// TwinCAT 3 PLC project Magnet_Measurement
// ProgramVersion: 3.1.4023.0
// libraries:
//   CmpBitmapPool, * (System)
//   Tc2_ControllerToolbox, * (Beckhoff Automation GmbH)
//   Tc2_Database, * (Beckhoff Automation GmbH)
//   Tc2_Standard, * (Beckhoff Automation GmbH)
//   Tc2_System, * (Beckhoff Automation GmbH)
//   Tc2_Utilities, * (Beckhoff Automation GmbH)
//   Tc3_Database, * (Beckhoff Automation GmbH)
//   Tc3_EventLogger, * (Beckhoff Automation GmbH)
//   Tc3_Module, * (Beckhoff Automation GmbH)
//   VisuDialogs, * (System)
//   VisuSymbols,3.5.10.0,System
// project tree:
//   DUTs/ ST_Data.TcDUT, ST_HMI_Plot_Array.TcDUT, ST_Masurdata.TcDUT, ST_Metadata.TcDUT
//   / GlobalTextList.TcGTLO, PlcTask.TcTTO, Visualisierungsmanager.TcVMO (not stored)
//   GVLs/ GVL_masur.TcGVL, GVL_IO.TcGVL, GVL_Meta.TcGVL
//   POUs/ FB_Write_Metadata.TcPOU, Log_Data_Buffer.TcPOU
//   VISUs/ GVL_Visu.TcGVL, ImagePool.TcIPO (not stored), Startpage.TcVIS, Write_Metadata_Visu.TcVIS, Visualization.TcVIS
// real-time tasks:
//   TASK PlcTask: cycle T#20ms, priority 20, ADS port 350
// I/O:
//   DEVICE Gerät 1 (EtherCAT) (disabled), AmsNetId 192.168.56.1.2.1
//     Box 1 (BK1120)

CONFIGURATION Magnet_Measurement
    RESOURCE PLC ON TwinCAT3
        TASK PlcTask(INTERVAL := T#20ms, PRIORITY := 20);
        PROGRAM Log_Data_Buffer WITH PlcTask : Log_Data_Buffer;
    END_RESOURCE
END_CONFIGURATION

// ---- DUTs/ST_Data.TcDUT
TYPE ST_Data :
STRUCT
	power: REAL;
	test: REAL;
	timestamp: REAL;
END_STRUCT
END_TYPE

// ---- DUTs/ST_HMI_Plot_Array.TcDUT
TYPE ST_HMI_Plot_Array :
STRUCT
	x : REAL := 0;
	y : REAL := 0;
END_STRUCT
END_TYPE

// ---- DUTs/ST_Masurdata.TcDUT
TYPE ST_Masurdata :
STRUCT
	id: INT;
	time2: REAL;
	primary_power: REAL;
	secondary_power: REAL;
	phase_shift: REAL;
	frequency: REAL;
	flux_density: REAL;
	Meta_id: INT;
END_STRUCT
END_TYPE

// ---- DUTs/ST_Metadata.TcDUT
TYPE ST_Metadata :
STRUCT
	Id: LINT;
	measurementname: STRING(255);
	carried_out: STRING(255);
	thickness: REAL;
	steel: STRING(255);
	joint_pre: STRING(255);
	root_face: REAL;
	opening_angel: REAL;
	edge_pre: STRING(255);
	welding_speed: REAL;
	laser_power: REAL;
	focal_position: REAL;
	distance_a_l: REAL;
	wire_feeding_rate: REAL;
	wire_diameter: REAL;
	wire_type: STRING(255);
	stickout: REAL;
	arc_dynamic: REAL;
	frequency: REAL;
	voltage_ac_power_source: REAL;
	distance_magnet_pole: REAL;
	magnet_pole_width: REAL;
	magnet_pole_type: STRING(255);
	core_dimension: REAL;
	very_good: STRING(255);
	normal: STRING(255);
	uniform_root_overcome: STRING(255);
	undercut: STRING(255);
	sporadic_seam_collapse: STRING(255);
	sporadic_dropout: STRING(255);
	bad: STRING(255);
	periodic_dropout: STRING(255);
	strong_seam_collapse: STRING(255);
	incomplite_penetration: STRING(255);
END_STRUCT
END_TYPE

// ---- GVLs/GVL_masur.TcGVL
{attribute 'qualified_only'}
VAR_GLOBAL
	id : INT; //wird automatisch erstellt
	time2 : REAL;
	primary_power: REAL;
	secondary_power: REAL;
	phase_shift: REAL;
	frequency: REAL;
	flux_density: REAL;
	Meta_id: INT;
END_VAR

// ---- GVLs/GVL_IO.TcGVL
{attribute 'qualified_only'}
VAR_GLOBAL
	//Raw data read every cycle
	//Primärspule
	gl_voltage_effective_raw_prime AT %I* : UINT := 15000; //Effektivwert Spannung Primärspule Rohwert
	gl_voltage_periode_raw_prime AT  %I* : UINT := 20; //Periode Spannungsignal Primärspule Rohwert
	gl_current_effective_raw_prime AT %I* : UINT := 3800; //Effektivwert Stromstärke Primärspule Rohwert
	gl_current_periode_raw_prime AT %I* : UINT := 20; //Periode Stromstärkesignal Primärspule Rohwert
	//Sekundärspule
	gl_voltage_effective_raw_secondary AT %I* : UINT := 20546; //Effektivwert Spannung Sekundärspule Rohwert
	gl_voltage_periode_raw_secondary AT  %I* : UINT := 20; //Periode Spannungsignal Sekundärspule Rohwert
	gl_current_effective_raw_secondary AT %I* : UINT := 3800; //Effektivwert Stromstärke Sekundärspule Rohwert
	gl_current_periode_raw_secondary AT %I* : UINT := 20; //Periode Stromstärkesignal Sekundärspule Rohwert
END_VAR

// ---- GVLs/GVL_Meta.TcGVL
{attribute 'qualified_only'}
VAR_GLOBAL
	// Variablen for Database Metadata Table
	Id : LINT := 11; //wird automatisch erstellt beim schreiben
	measurementname: STRING(255) := 'test';
	carried_out: STRING(255) := 'test1';
	thickness: REAL := 1;
	steel: STRING(255) := 'stahl';
	joint_pre: STRING(255) := 'squer';
	root_face: REAL := 0;
	opening_angel: REAL := 0;
	edge_pre: STRING(255) := 'aet';
	welding_speed: REAL := 0;
	laser_power: REAL := 1;
	focal_position: REAL := 2;
	distance_a_l: REAL := 3;
	wire_feeding_rate: REAL := 4;
	wire_diameter: REAL := 5;
	wire_type: STRING(255) := 'tea';
	stickout: REAL := 6;
	arc_dynamic: REAL := 2;
	frequency: REAL := 1;
	voltage_ac_power_source: REAL := 22;
	distance_magnet_pole: REAL := 33;
	magnet_pole_width: REAL := 22;
	magnet_pole_type: STRING(255) := 'at';
	core_dimension: REAL := 22;
	very_good: STRING(255) := 'asd';
	normal: STRING(255) := 'asd';
	uniform_root_overcome: STRING(255) := 'asd';
	undercut: STRING(255) := 'asdw';
	sporadic_seam_collapse: STRING(255) := 'aaa';
	sporadic_dropout: STRING(255) := 'aw';
	bad: STRING(255) := 'aaaw';
	periodic_dropout: STRING(255) := 'asdaw';
	strong_seam_collapse: STRING(255) := 'aqqq';
	incomplite_penetration: STRING(255) := 'öpkl';
END_VAR

// ---- VISUs/GVL_Visu.TcGVL
{attribute 'qualified_only'}
VAR_GLOBAL
	start_record : BOOL := FALSE;
END_VAR

// ---- POUs/Log_Data_Buffer.TcPOU
PROGRAM Log_Data_Buffer
VAR
	//Messvariablen
	voltage_effective_prime : REAL; //Effektivwert Spannung Primärspule umgewandelt auf +-10V
	voltage_frequency_prime : REAL; //Frequenz Primärspule Spannungssignal umgewandelt auf +-10 in Hz
	current_effective_prime : REAL; //Effektivwert Stromstärke Primärspule umgewandelt auf +-10V umgewandelt zu Ampere
	current_frequency_prime : REAL; //Frequenz Primärspule Stromstärkesignal umgewandelt auf +-10 Hz
	voltage_effective_secondary : REAL; //Effektivwert Spannung Sekundärspule umgewandelt auf +-10V
	voltage_frequency_secondary : REAL; //Frequenz Sekundärspule Spannungssignal umgewandelt auf +-10 Hz
	current_effective_secondary : REAL; //Effektivwert Stromstärke Sekundärspule umgewandelt auf +-10V umgewandelt zu Ampere
	current_frequency_secondary : REAL; //Frequenz Sekundärspule Stromstärkesignal umgewandelt auf +-10 Hz
	power_prime : REAL; //Leistung Primärspule W
	power_secondary : REAL; //Leistung Sekundärspule W
    
	//Arrays zum Plotten für HMI
	power_hmi_array : ARRAY[1..2,1..100] OF ST_HMI_Plot_Array;
	//power_secondary_hmi_array : ARRAY[1..1,1..100] OF ST_HMI_Plot_Array;
	i : INT := 1;
    rand : DRAND; 
    nrand: LREAL;
	
	fbGetCurTaskIdx  : GETCURTASKINDEX;
    ncycletime       : REAL;
	nState: INT;	
	bRecord : BOOL;
	//for generating timestamp
	fbGetSystemTime1: GetSystemTime;
	dwTimeLoDW: DWORD;
	dwTimeHiDW: DWORD;
	tFileTime: T_FILETIME;
	nTimestamp: REAL;
	//for insert meta data
	fbWriteMetadata : FB_Write_Metadata;
	fb_Start_Log : FB_PLCDBAutoLogEvt (sNetID:='', tTimeout := T#1S);
	write_meta : BOOL;
	write_meta_status : BOOL; 
	write_meta_error : BOOL; 
	meta_data_written_index : INT := 1;
	
	//for insert masur samples
	fbPLCDBCmd: FB_PLCDBCmdEvt(sNetID:= '', tTimeout:= T#19S);
	aPara: ARRAY [0..7] OF ST_ExpParameter;	
	sCmd1: STRING(255);
	sCmd2: STRING(255);
	sCmd: STRING(512); //CONCAT of sCmd1 and sCmd2
	
	//Data buffer for masur data
	aWriteSQL: ARRAY [0..19] OF BOOL;
	stData: ARRAY [0..19,0..99] OF ST_Masurdata;
	
	//buffer index and masur data variables
	nWriteBufferIndex: INT := 0;
	nWriteIndex: INT := 0;
	nSQLIndex: INT := 0;					
	bError: BOOL;
	bTableCreated: BOOL;
	bRecording: BOOL;
	nRecords: INT;
	sTableName: T_MaxString := 'masur';
	nDBID: UDINT := 1;
	timestampp : REAL := 0;
	index : INT := 0;
	id: INT := 1852;
	
	// Eventlogger
	ipTcResult: Tc3_Database.I_TcMessage;

END_VAR

// Convert Data and get the raw data
//Primärspule
rand();
nrand := rand.Num;
voltage_effective_prime := UINT_TO_REAL(GVL_IO.gl_voltage_effective_raw_prime)/65535*20; //Map UINT range of 0:65535 to +-10V 
voltage_frequency_prime := 1/(UINT_TO_REAL(GVL_IO.gl_voltage_periode_raw_prime)/1000); //convert ms to S and get Frequency from Period
current_effective_prime := UINT_TO_REAL(GVL_IO.gl_current_effective_raw_prime)/65535*20; //Map UINT range of 0:65535 to +-10V 
current_frequency_prime := 1/(UINT_TO_REAL(GVL_IO.gl_current_periode_raw_prime)/1000); //convert ms to S and get Frequency from Period
power_prime := voltage_effective_prime * current_effective_prime + nrand/3;
//Sekundärspule
voltage_effective_secondary := UINT_TO_REAL(GVL_IO.gl_voltage_effective_raw_secondary)/65535*20; //Map UINT range of 0:65535 to +-10V 
voltage_frequency_secondary := 1/(UINT_TO_REAL(GVL_IO.gl_voltage_periode_raw_secondary)/1000); //convert ms to S and get Frequency from Period
current_effective_secondary := UINT_TO_REAL(GVL_IO.gl_current_effective_raw_secondary)/65535*20; //Map UINT range of 0:65535 to +-10V 
current_frequency_secondary := 1/(UINT_TO_REAL(GVL_IO.gl_current_periode_raw_secondary)/1000); //convert ms to S and get Frequency from Period
power_secondary := voltage_effective_secondary * current_effective_secondary + nrand/2;

fbGetCurTaskIdx();
ncycletime := _TaskInfo[fbGetCurTaskIdx.index].CycleTime/10000;

//HMI Plot Array befüllen
IF (i <= 100) THEN
	//power_prime_hmi_array[1,i].x := i*ncycletime;
	//power_prime_hmi_array[1,i].y := power_prime;
	//power_secondary_hmi_array[1,i].x := i*ncycletime;
	//power_secondary_hmi_array[1,i].y := power_secondary;
	power_hmi_array[1,i].x := i*ncycletime;
	power_hmi_array[1,i].y := power_prime;
	power_hmi_array[2,i].x := i*ncycletime;
	power_hmi_array[2,i].y := power_secondary;
	i := i +1;
	ELSE
		i := 1;
END_IF
//FOR i := 1 TO 100 DO
//	power_prime_hmi_array[1,i].x := i;
//	power_prime_hmi_array[1,i].x := i;
//END_FOR//

//Create timestamp
fbGetSystemTime1(timeLoDW=>dwTimeLoDW,timeHiDW=>dwTimeHiDW);
tFileTime.dwLowDateTime := dwTimeLoDW;
tFileTime.dwHighDateTime := dwTimeHiDW;	
MEMCPY(ADR(nTimestamp), ADR(tFileTime), 8);

CASE nState OF
	0://Init
		IF bRecord THEN			
			bError := FALSE;
			bRecording := FALSE;
			nRecords := 0;
			//sTableName := 'Magnet';//CONCAT('tbl_TestSignals_', LINT_TO_STRING(nTimestamp)); //create new tablename
			sCmd1 := CONCAT('INSERT INTO ', sTableName);
			sCmd2 := ' ([id],[time2],[primary_power],[secondary_power],[phase_shift],[frequency],[flux_density],[Meta_id]) VALUES({id},{time2},{primary_power},{secondary_power},{phase_shift},{frequency},{flux_density},{Meta_id});';
			CONCAT2(ADR(sCmd1), ADR(sCmd2), ADR(sCmd), SIZEOF(sCmd));
			
			aPara[0].sParaName:= 'id'; 				aPara[0].nParaSize:= 8; 	aPara[0].eParaType:= E_ExpParameterType.Int32 ;
			aPara[1].sParaName:= 'time2'; 			aPara[1].nParaSize:= 8; 	aPara[1].eParaType:= E_ExpParameterType.Float32 ;		
			aPara[2].sParaName:= 'primary_power';	aPara[2].nParaSize:= 8;		aPara[2].eParaType:= E_ExpParameterType.Float32 ;		
			aPara[3].sParaName:= 'secondary_power';	aPara[3].nParaSize:= 8;		aPara[3].eParaType:= E_ExpParameterType.Float32 ;	
			aPara[4].sParaName:= 'phase_shift';		aPara[4].nParaSize:= 8;		aPara[4].eParaType:= E_ExpParameterType.Float32 ;
			aPara[5].sParaName:= 'frequency';		aPara[5].nParaSize:= 8;		aPara[5].eParaType:= E_ExpParameterType.Float32 ;
			aPara[6].sParaName:= 'flux_density';	aPara[6].nParaSize:= 8;		aPara[6].eParaType:= E_ExpParameterType.Float32 ;
			aPara[7].sParaName:= 'Meta_id';			aPara[7].nParaSize:= 8;		aPara[7].eParaType:= E_ExpParameterType.Int32 ;	
			nWriteBufferIndex := 0;
			nWriteIndex := 0;
			nSQLIndex := 0;	
			nState := 1;
		END_IF
		
	1://Idle
		IF write_meta THEN
			IF meta_data_written_index = 1 THEN
				fb_Start_Log.RunOnce(hAutologGrpID := 1, bAll := TRUE);
				meta_data_written_index := 2;
			ELSE 
				fb_Start_Log.RunOnce(hAutologGrpID := 1, bAll := TRUE);
				fb_Start_Log.RunOnce(hAutologGrpID := 1, bAll := TRUE);
				fb_Start_Log.RunOnce(hAutologGrpID := 1, bAll := TRUE);
			END_IF
			write_meta := FALSE;
			write_meta_status := fb_Start_Log.bBusy;
			write_meta_error := fb_Start_Log.bError;
		END_IF
		
	2://Recording		
		bRecording := TRUE;
		//Fill buffer
		stData[nWriteBufferIndex, nWriteIndex].id := id;
		stData[nWriteBufferIndex, nWriteIndex].time2 := timestampp;
		stData[nWriteBufferIndex, nWriteIndex].primary_power := power_prime;
		stData[nWriteBufferIndex, nWriteIndex].secondary_power := power_secondary;
		stData[nWriteBufferIndex, nWriteIndex].phase_shift := 1.0;
		stData[nWriteBufferIndex, nWriteIndex].frequency := 2.0;
		stData[nWriteBufferIndex, nWriteIndex].flux_density := 3.0;
		stData[nWriteBufferIndex, nWriteIndex].Meta_id := 1;
		timestampp := ncycletime * index;
		index := index + 1;
		id := id + 1;
		//Set buffer index
		nWriteIndex := nWriteIndex + 1;		
		IF nWriteIndex = 100 THEN
			nWriteIndex := 0;
			aWriteSQL[nWriteBufferIndex]:= TRUE;
			nWriteBufferIndex := nWriteBufferIndex + 1;
			
			IF nWriteBufferIndex = 20 THEN
				nWriteBufferIndex := 0;
			END_IF 	
			
			IF aWriteSQL[nWriteBufferIndex] THEN
				nState := 255;
				RETURN;
			END_IF
		END_IF
				
		//Write buffer element (100 samples) to database
		IF aWriteSQL[nSQLIndex] THEN
			ipTcResult := fbPLCDBCmd.ipTcResult;
			IF fbPLCDBCmd.Execute(nDBID, ADR(sCmd), SIZEOF(sCmd), ADR(stData[nSQLIndex,0]), SIZEOF(stData[nSQLIndex,0]) * 100, ADR(aPara), SIZEOF(aPara)) THEN
				IF fbPLCDBCmd.bError THEN					
					nState := 255;
				ELSE
					nRecords := nRecords + 100;
					
					aWriteSQL[nSQLIndex] := FALSE;
					
					nSQLIndex := nSQLIndex + 1;
					IF nSQLIndex = 20 THEN
						nSQLIndex := 0;
					END_IF
					
					IF NOT bRecord THEN
						bRecording := FALSE;
						nState := 0;
					END_IF
				END_IF				
			END_IF
		END_IF
		
	255://Error
		bError := TRUE;
		bRecording := FALSE;
		IF NOT bRecord THEN			
			nState := 0;
		END_IF 
END_CASE

END_PROGRAM

// ---- POUs/FB_Write_Metadata.TcPOU
FUNCTION_BLOCK FB_Write_Metadata
VAR
	stMetadata : ST_Metadata;
	//fbPLCWrite : FB_PLCDBWriteEvt(sNetID:='', tTimeout:=T#15S);
	//arrColumns: ARRAY[0..33] OF STRING(255) := ['Id', 'measurementname', 'carried_out', 'thickness', 'steel', 'joint_pre', 'root_face', 'opening_angel', 'edge_pre', 'welding_speed', 'laser_power', 'focal_position', 'distance_a_l', 'wire_feeding_rate', 'wire_diameter', 'wire_type', 'stickout', 'arc_dynamic', 'frequency', 'voltage_ac_power_source', 'distance_magnet_pole', 'magnet_pole_width', 'magnet_pole_type', 'core_dimension', 'very_good', 'normal', 'uniform_root_overcome', 'undercut', 'sporadic_seam_collapse', 'sporadic_dropout', 'bad', 'periodic_dropout', 'strong_seam_collapse', 'incomplite_penetration'];
	stData123 : ST_Data;
	fb_PLCDBWriteEvt: FB_PLCDBWriteEvt(sNetID:='', tTimeout:=T#5S);
	arrColumns: ARRAY [0..2] OF STRING(50) := ['power', 'test', 'timestamp'];
	
END_VAR
VAR_OUTPUT
	status : BOOL;
END_VAR

// Get variables from global list form Visu Interface 
stMetadata.Id := GVL_Meta.Id;
stMetadata.measurementname := GVL_Meta.measurementname;
stMetadata.carried_out := GVL_Meta.carried_out;
stMetadata.thickness := GVL_Meta.thickness;
stMetadata.steel := GVL_Meta.steel;
stMetadata.joint_pre := GVL_Meta.joint_pre;
stMetadata.root_face := GVL_Meta.root_face;
stMetadata.opening_angel := GVL_Meta.opening_angel;
stMetadata.edge_pre := GVL_Meta.edge_pre;
stMetadata.welding_speed := GVL_Meta.welding_speed;
stMetadata.laser_power := GVL_Meta.laser_power;
stMetadata.focal_position := GVL_Meta.focal_position;
stMetadata.distance_a_l := GVL_Meta.distance_a_l;
stMetadata.wire_feeding_rate := GVL_Meta.wire_feeding_rate;
stMetadata.wire_diameter := GVL_Meta.wire_diameter;
stMetadata.wire_type := GVL_Meta.wire_type;
stMetadata.stickout := GVL_Meta.stickout;
stMetadata.arc_dynamic := GVL_Meta.arc_dynamic;
stMetadata.frequency := GVL_Meta.frequency;
stMetadata.voltage_ac_power_source := GVL_Meta.voltage_ac_power_source;
stMetadata.distance_magnet_pole := GVL_Meta.distance_magnet_pole;
stMetadata.magnet_pole_width := GVL_Meta.magnet_pole_width;
stMetadata.magnet_pole_type := GVL_Meta.magnet_pole_type;
stMetadata.core_dimension := GVL_Meta.core_dimension;
stMetadata.very_good := GVL_Meta.very_good;
stMetadata.normal := GVL_Meta.normal;
stMetadata.uniform_root_overcome := GVL_Meta.uniform_root_overcome;
stMetadata.undercut := GVL_Meta.undercut;
stMetadata.sporadic_seam_collapse := GVL_Meta.sporadic_seam_collapse;
stMetadata.sporadic_dropout := GVL_Meta.sporadic_dropout;
stMetadata.bad := GVL_Meta.bad;
stMetadata.periodic_dropout := GVL_Meta.periodic_dropout;
stMetadata.strong_seam_collapse := GVL_Meta.strong_seam_collapse;
stMetadata.incomplite_penetration := GVL_Meta.incomplite_penetration;

//Test
stData123.power := 1.0;
stData123.test := 2.0;
stData123.timestamp := 3.0;
//IF NOT fb_PLCDBWriteEvt.bBusy THEN
	fb_PLCDBWriteEvt.WriteStruct(
			hDBID:= 1, 
			sTableName:= 'Magnet', 
			pRecord:= ADR(stData123), 
			cbRecord:= SIZEOF(stData123), 
			pColumnNames:= ADR(arrColumns), 
			cbColumnNames:= SIZEOF(arrColumns));
//END_IF

//write struct with event to database table Meta
//IF NOT fbPLCWrite.bBusy THEN
//	fbPLCWrite.WriteStruct(
//	hDBID:= 1, 
//	sTableName:= 'Meta', 
//	pRecord:= ADR(stMetadata), 
//	cbRecord:= SIZEOF(stMetadata), 
//	pColumnNames:= ADR(arrColumns), 
//	cbColumnNames:= SIZEOF(arrColumns));
//END_IF

//IF fbPLCWrite.bError THEN
//	status := TRUE;
//ELSE
//	status := FALSE;	
//END_IF

END_FUNCTION_BLOCK

// ---- GlobalTextList.TcGTLO
TEXTLIST GlobalTextList
  699 = '%f'
  92 = '%i'
  962 = '%s'
  908 = 'Arc Dynamic'
  755 = 'Bad'
  149 = 'Carried Out'
  470 = 'Core Dimension'
  79 = 'Distance a_l'
  864 = 'Distance Magnet Pole'
  103 = 'dtj'
  832 = 'Edge Pre'
  480 = 'est'
  342 = 'Focal Position'
  478 = 'Frequency'
  55 = 'ID'
  734 = 'Incomplete Penetration'
  457 = 'Joint Pre'
  502 = 'Laser Power'
  766 = 'Magent Pole Type'
  266 = 'Magnet Measurement HMI'
  930 = 'Magnet Pole Width'
  422 = 'Measurement\t Name'
  335 = 'Measurement Name'
  56 = 'Measurementname'
  340 = 'Measurmentname'
  418 = 'Normal'
  193 = 'Opening Angel'
  887 = 'Periodic Dopout'
  9 = 'Root Face'
  388 = 'Root Opening Angel'
  257 = 'Sporadic Dropout'
  200 = 'Sporadic Seam Collapse'
  327 = 'Start PLC Connection'
  42 = 'Status'
  144 = 'Statusword'
  188 = 'Steel'
  46 = 'Stickout'
  650 = 'Strong Seam Collapse'
  230 = 'Thickness'
  58 = 'Undercut'
  974 = 'Uniform Root Overcome'
  95 = 'Very Good'
  336 = 'Voltafage AC Power Source'
  711 = 'Voltage AC Power Source'
  745 = 'Voltatage AC Power Source'
  341 = 'Welding Speed'
  262 = 'WER'
  106 = 'Wire Diameter'
  270 = 'Wire Feeding Rate'
  572 = 'Wire Type'
  182 = 'Write Metadata'
END_TEXTLIST

// ---- VISUs/Startpage.TcVIS
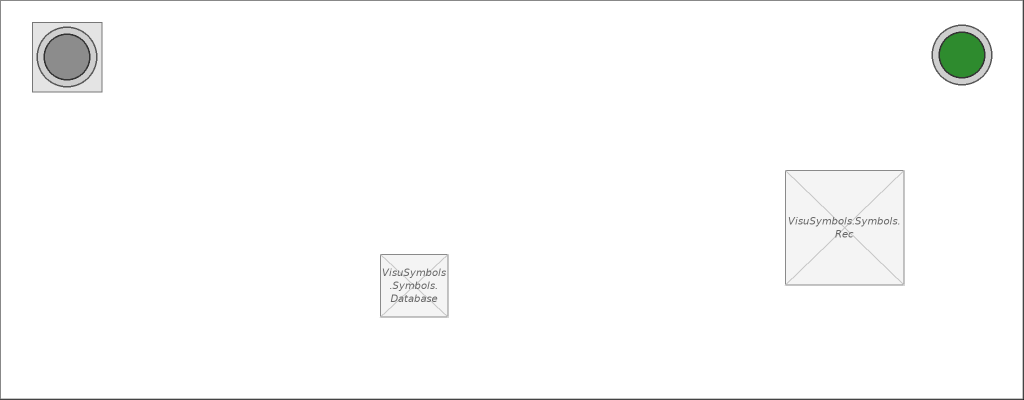
VISUALIZATION Startpage  // 1024x400
    RoundedRectangle (0,0 1024x400)
    PushSwitchLed (32,22 70x70), behaviour: TOGGLE, style: Switch-PushSwitchLed-Gray
    Lamp1 (927,20 70x70), style: Lamp-Lamp1-Green
    Image (785,170 119x115), image: VisuSymbols.Symbols.Rec
    Image (380,254 68x63), image: VisuSymbols.Symbols.Database
END_VISUALIZATION

// ---- VISUs/Write_Metadata_Visu.TcVIS
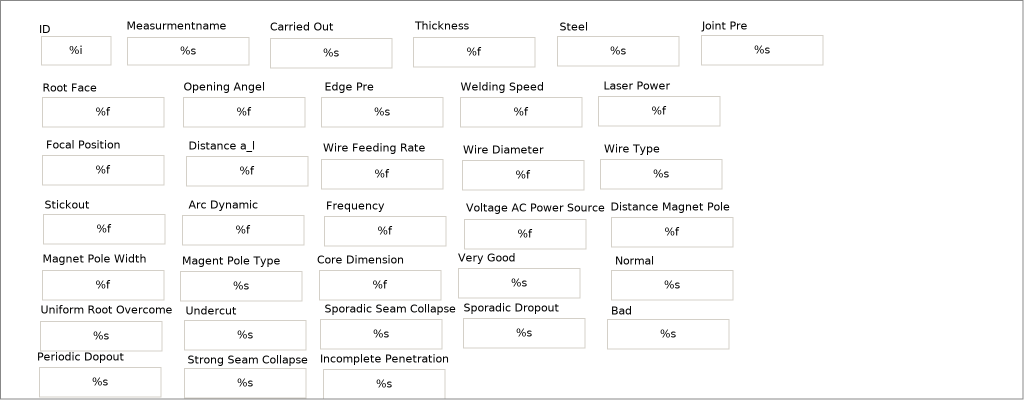
VISUALIZATION Write_Metadata_Visu  // 1024x400
    Textfield (41,36 70x29), "%i", text variable: GVL_Meta.Id
        OnMouseDown: write the text variable via Default
    Label (10,15 70x29), "ID"
    Textfield (127,37 122x28), "%s", text variable: GVL_Meta.measurementname
        OnMouseClick: write the text variable via Default
    Label (117,13 119x26), "Measurmentname"
    Textfield (270,38 122x30), "%s", text variable: GVL_Meta.Id
        OnMouseClick: write the text variable via Default
    Label (264,13 76x28), "Carried Out"
    Textfield (413,37 122x30), "%f", text variable: GVL_Meta.thickness
        OnMouseClick: write the text variable via Default
    Label (404,12 76x28), "Thickness"
    Textfield (557,36 122x30), "%s", text variable: GVL_Meta.steel
        OnMouseClick: write the text variable via Default
    Label (545,13 58x28), "Steel"
    Textfield (701,35 122x30), "%s", text variable: GVL_Meta.joint_pre
        OnMouseClick: write the text variable via Default
    Label (696,12 58x28), "Joint Pre"
    Textfield (42,97 122x30), "%f", text variable: GVL_Meta.root_face
        OnMouseClick: write the text variable via Default
    Label (41,74 58x28), "Root Face"
    Textfield (183,97 122x30), "%f", text variable: GVL_Meta.opening_angel
        OnMouseClick: write the text variable via Default
    Label (167,73 115x28), "Opening Angel"
    Textfield (321,97 122x30), "%s", text variable: GVL_Meta.edge_pre
        OnMouseClick: write the text variable via Default
    Label (316,73 67x28), "Edge Pre"
    Textfield (460,97 122x30), "%f", text variable: GVL_Meta.welding_speed
        OnMouseClick: write the text variable via Default
    Label (451,73 103x28), "Welding Speed"
    Textfield (598,96 122x30), "%f", text variable: GVL_Meta.laser_power
        OnMouseClick: write the text variable via Default
    Label (588,72 98x28), "Laser Power"
    Textfield (42,155 122x30), "%f", text variable: GVL_Meta.focal_position
        OnMouseClick: write the text variable via Default
    Label (26,131 115x28), "Focal Position"
    Textfield (186,156 122x30), "%f", text variable: GVL_Meta.distance_a_l
        OnMouseClick: write the text variable via Default
    Label (173,132 98x28), "Distance a_l"
    Textfield (321,159 122x30), "%f", text variable: GVL_Meta.wire_feeding_rate
        OnMouseClick: write the text variable via Default
    Label (317,134 115x28), "Wire Feeding Rate"
    Textfield (462,160 122x30), "%f", text variable: GVL_Meta.wire_diameter
        OnMouseClick: write the text variable via Default
    Label (446,136 115x28), "Wire Diameter"
    Textfield (600,159 122x30), "%s", text variable: GVL_Meta.wire_type
        OnMouseClick: write the text variable via Default
    Label (589,135 86x28), "Wire Type"
    Textfield (43,214 122x30), "%f", text variable: GVL_Meta.stickout
        OnMouseClick: write the text variable via Default
    Label (33,191 68x28), "Stickout"
    Textfield (182,215 122x30), "%f", text variable: GVL_Meta.arc_dynamic
        OnMouseClick: write the text variable via Default
    Label (166,191 115x28), "Arc Dynamic"
    Textfield (324,216 122x30), "%f", text variable: GVL_Meta.frequency
        OnMouseClick: write the text variable via Default
    Label (298,192 115x28), "Frequency"
    Textfield (464,219 122x30), "%f", text variable: GVL_Meta.voltage_ac_power_source
        OnMouseClick: write the text variable via Default
    Label (454,194 163x28), "Voltage AC Power Source"
    Textfield (611,217 122x30), "%f", text variable: GVL_Meta.distance_magnet_pole
        OnMouseClick: write the text variable via Default
    Label (603,193 135x28), "Distance Magnet Pole"
    Textfield (42,270 122x30), "%f", text variable: GVL_Meta.magnet_pole_width
        OnMouseClick: write the text variable via Default
    Label (37,245 115x28), "Magnet Pole Width"
    Textfield (180,271 122x30), "%s", text variable: GVL_Meta.magnet_pole_type
        OnMouseClick: write the text variable via Default
    Label (174,247 115x28), "Magent Pole Type"
    Textfield (319,270 122x30), "%f", text variable: GVL_Meta.core_dimension
        OnMouseClick: write the text variable via Default
    Label (303,246 115x28), "Core Dimension"
    Textfield (458,268 122x30), "%s", text variable: GVL_Meta.very_good
        OnMouseClick: write the text variable via Default
    Label (440,244 94x28), "Very Good"
    Textfield (611,270 122x30), "%s", text variable: GVL_Meta.normal
        OnMouseClick: write the text variable via Default
    Label (601,247 67x28), "Normal"
    Textfield (40,321 122x30), "%s", text variable: GVL_Meta.uniform_root_overcome
        OnMouseClick: write the text variable via Default
    Label (32,296 149x28), "Uniform Root Overcome"
    Textfield (184,320 122x30), "%s", text variable: GVL_Meta.undercut
        OnMouseClick: write the text variable via Default
    Label (172,297 78x28), "Undercut"
    Textfield (320,319 122x30), "%s", text variable: GVL_Meta.sporadic_seam_collapse
        OnMouseClick: write the text variable via Default
    Label (315,295 151x28), "Sporadic Seam Collapse"
    Textfield (463,318 122x30), "%s", text variable: GVL_Meta.sporadic_dropout
        OnMouseClick: write the text variable via Default
    Label (454,294 115x28), "Sporadic Dropout"
    Textfield (607,319 122x30), "%s", text variable: GVL_Meta.bad
        OnMouseClick: write the text variable via Default
    Label (589,297 65x28), "Bad"
    Textfield (39,367 122x30), "%s", text variable: GVL_Meta.periodic_dropout
        OnMouseClick: write the text variable via Default
    Label (23,343 115x28), "Periodic Dopout"
    Textfield (184,368 122x30), "%s", text variable: GVL_Meta.strong_seam_collapse
        OnMouseClick: write the text variable via Default
    Label (180,346 136x28), "Strong Seam Collapse"
    Textfield (323,369 122x30), "%s", text variable: GVL_Meta.incomplite_penetration
        OnMouseClick: write the text variable via Default
    Label (307,345 155x28), "Incomplete Penetration"
END_VISUALIZATION

// ---- VISUs/Visualization.TcVIS
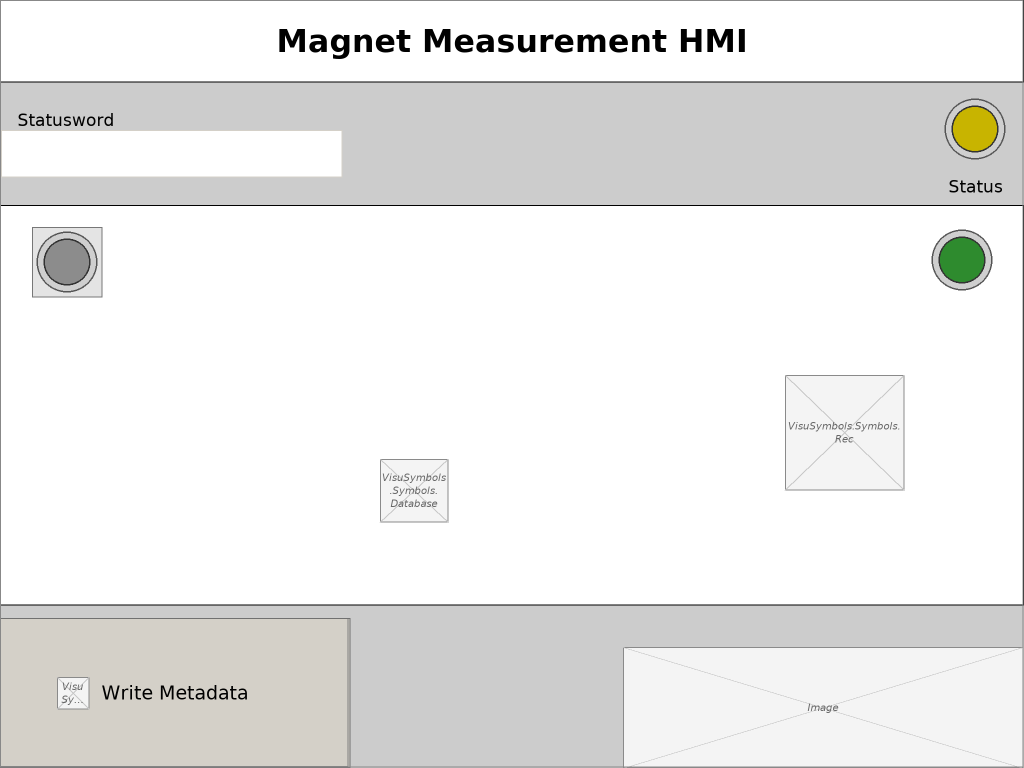
VISUALIZATION Visualization  // 1024x768
    Button (0,618 350x150), "Write Metadata"
        OnMouseClick: FrameSelectionChange Selection=SelectedFrame=f10d8547-6667-49de-9f33-336b6c15e565, Selection=1, GlobSel=AssignType=Directly, SelType=Locally
    RoundedRectangle (0,0 1024x82), "Magnet Measurement HMI"
    Image (623,647 400x121)
        p84334746: 'BAM_Logo'
    Lamp1 (940,94 70x70), tooltip "Status", style: Lamp-Lamp1-Yellow
    Label (941,167 70x39), "Status"
    Frame (0,205 1024x400)
        shows Startpage()
        shows Write_Metadata_Visu()
    Textfield (1,130 341x47)
    Label (5,105 122x30), "Statusword"
    Image (57,677 32x32), image: VisuSymbols.Symbols.Edit
END_VISUALIZATION
